(* CODESYS project FU_dwBitPart.xml

Project tree, tasks and I/O mapping:
  function FU_dwBitPart [ST]
*)

// FU_dwBitPart
//This function changed only the needed bits of a variable
// |**Version**|**Author**| **Date** |**Changes**
// | 1         | NSN      | 16-03-22 | Creation
FUNCTION FU_dwBitPart : BOOL
VAR_IN_OUT
	valueChange		:DWORD;		//Variable to change
END_VAR
VAR_INPUT
	value			:DWORD;		//Value to change bits to
	amount			:BYTE;		//Amount of bits to change
	offset			:BYTE;		//Offset in variable to change bits at
END_VAR

valueChange		:=		(valueChange AND ROL(GConstants.binaryInvMaskDWord[amount],offset)) OR SHL(value AND GConstants.binaryMaskDWord[amount],offset);

END_FUNCTION
